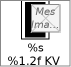
VISUALIZATION VISU_ALIM_HT  // 71x67
VAR_IN_OUT
	m_Input_HT:				BLOCK_HT_CANON_ST10;
END_VAR
VAR_IN_OUT
	m_Input_NO_HV_RET:		BOOL;
END_VAR
    Rectangle (25,2 20x35), colour toggle: m_Input_HT.STATE_HV_ON, invisible if: NOT m_Input_HT.STATE_HV_ON AND NOT m_Input_HT.STATE_HV
    Rectangle (25,2 20x35), invisible if: m_Input_HT.STATE_HV_ON OR m_Input_HT.STATE_HV
    Polygon (41,73)
    Rectangle (21,0 28x39), invisible if: NOT m_Input_HT.HV.AUTOR_On_IHM AND NOT m_Input_HT.HV.AUTOR_Off_IHM, input disabled if: (NOT m_Input_HT.HV.AUTOR_ON_IHM AND NOT m_Input_HT.HV.AUTOR_OFF_IHM) OR NOT PRG_User.ACTU_USER.MAINTENANCE
        tap m_Input_HT.HV.M_On
    Rectangle (0,41 71x14), "%s", text variable: m_Input_HT.MNEMO
    Rectangle (0,55 71x12), "%1.2f KV", text variable: m_Input_HT.STATE_V_HV, invisible if: (m_Input_NO_HV_RET) <> 0
    Image (31,4 29x28), invisible if: NOT m_Input_HT.STATE_NOK, image: MesImages.warning
END_VISUALIZATION

(* stored: Version 1.1.0.1, ProductVersion 3.1.4024.10
   Visu VISU_ALIM_HT: Id {827967d0-8ca9-4ddd-a382-bde073527560} *)
